PROGRAM prgInputMapp
VAR
END_VAR

;

END_PROGRAM

(* stored: Version 1.1.0.1, ProductVersion 3.1.4026.18
   POU prgInputMapp: Id {99bd5eed-e25f-4710-b535-8567b88e1446}, SpecialFunc None *)
